FUNCTION_BLOCK IA_FPTO (* ISOBUS Adapter for Front Power Take off (FPTO) *)
  (* Standard: ISO 11783-7; Classification: PGN 65092; Description: Copyright (c) 2024-2026 HR Agrartechnik GmbH This program and the accompanying materials are made available under the terms of the Eclipse Public License 2.0 which is available at https://www.eclipse.org/legal/epl-2.0/ SPDX-License-Identifier: EPL-2.0 *)
  (* Version 1.0, 2026-04-19, Franz Höpfinger, HR Agrartechnik GmbH, initial API and implementation (Adapter Wrapper for I_FPTO) *)
  PACKAGE isobus::tecu;
  IMPORT eclipse4diac::core::TypeHash;
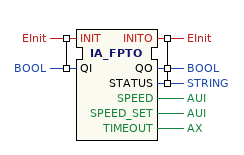
  EVENT_INPUT
    INIT : EInit WITH QI; (* Service Initialization *)
  END_EVENT
  EVENT_OUTPUT
    INITO : EInit WITH QO, STATUS; (* Initialization Confirm *)
  END_EVENT
  VAR_INPUT
    QI : BOOL; (* Event Input Qualifier *)
  END_VAR
  VAR_OUTPUT
    QO : BOOL; (* Event Output Qualifier *)
    STATUS : STRING;
  END_VAR
  PLUGS
    SPEED : adapter::types::unidirectional::AUI; (* Front PTO output shaft speed *)
    SPEED_SET : adapter::types::unidirectional::AUI; (* Front PTO output shaft speed set point *)
    TIMEOUT : adapter::types::unidirectional::AX; (* Timeout Status *)
  END_PLUGS
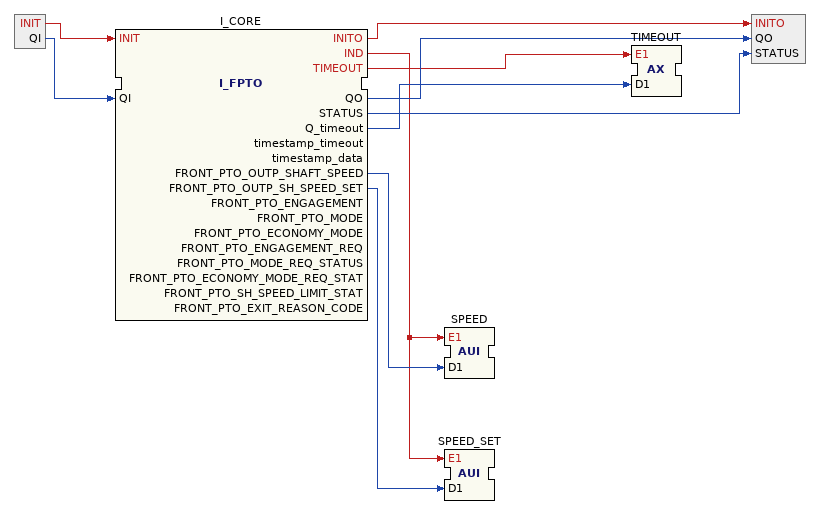
  FBS
    I_CORE : isobus::tecu::I_FPTO;
  END_FBS
  EVENT_CONNECTIONS
    INIT TO I_CORE.INIT;
    I_CORE.INITO TO INITO;
    I_CORE.IND TO SPEED.E1;
    I_CORE.IND TO SPEED_SET.E1;
    I_CORE.TIMEOUT TO TIMEOUT.E1;
  END_CONNECTIONS
  DATA_CONNECTIONS
    QI TO I_CORE.QI;
    I_CORE.QO TO QO;
    I_CORE.STATUS TO STATUS;
    I_CORE.FRONT_PTO_OUTP_SHAFT_SPEED TO SPEED.D1;
    I_CORE.FRONT_PTO_OUTP_SH_SPEED_SET TO SPEED_SET.D1;
    I_CORE.Q_timeout TO TIMEOUT.D1;
  END_CONNECTIONS
END_FUNCTION_BLOCK
